{attribute addProperty BoxType "AX5118-0000-0011-0011"}
{attribute addProperty Id "Drive_status_wordAT %I*UINT1620Position_feedback_1_valueAT %I*DINT3240"}
{attribute addProperty CRC "43974933"}
{attribute addProperty SizeInBites "48"}
{attribute addProperty SizeInBytes "6"}
TYPE AT_x_029F0115 :
STRUCT
	{attribute addProperty Name "Drive_status_word"}
	Drive_status_word AT %I* : UINT;
	{attribute addProperty Name "Position_feedback_1_value"}
	Position_feedback_1_value AT %I* : DINT;
END_STRUCT
END_TYPE

(* stored: Version 1.2.0.0, ProductVersion 3.1.4024.9
   DUT AT_x_029F0115: Id {38e68895-b093-444b-b356-0186900be683} *)
